FUNCTION_BLOCK Station1Control (* Basic FB with empty ECC *)
  (* Standard: 61499-2 *)
  (* Version 1.0, 2021-09-15, dorofeev *)
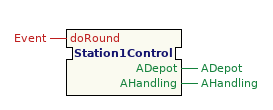
  EVENT_INPUT
    doRound;
  END_EVENT
  PLUGS
    ADepot : ADepot;
    AHandling : AHandling;
  END_PLUGS
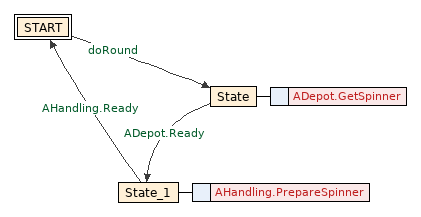
  EC_STATES
    START; (* Initial State *)
    State : -> ADepot.GetSpinner;
    State_1 : -> AHandling.PrepareSpinner;
  END_STATES
  EC_TRANSITIONS
    START TO State := doRound;
    State TO State_1 := ADepot.Ready;
    State_1 TO START := AHandling.Ready;
  END_TRANSITIONS
END_FUNCTION_BLOCK
